// SIMATIC S7-200 project (STEP 7-Micro/WIN), CPU 226 CN REL 02.01

SYMBOL_TABLE 用户定义1
系统年              VW1648
本班开始运行小时         VW1680
本班开始运行分钟         VW1684
本班开始运行秒          VW1688
本班运行日            VW3778
系统日              VW1652
系统秒              VW1664
EEPROM写入次数       VW3558
累计运行分钟           VW1624
EEPROM写入后对秒脉冲计   VW3368
累计运行小时           VW1620
EEPROM写入后计时      M30.1
EEPROM传送中        SM31.7
SA2              I0.0     // 联锁/单独(单独=0/联锁=1)
PH1              I0.1     // 第1段线体首光电开关
PH11             I0.2     // 第1段线体末光电开关
PH2              I0.3     // 第2段线体首光电开关
PH21             I0.4     // 第2段线体末光电开关
PH3              I0.5     // 第3段线体首光电开关
PH31             I0.6     // 第3段线体末光电开关
PH4              I0.7     // 第4段线体首光电开关
PH41             I1.0     // 第4段线体末光电开关
PH5              I1.1     // 第5段线体首光电开关
PH6              I1.2     // 第6段线体末光电开关
PH7              I1.3     // 第7段线体首光电开关
PH71             I1.4     // 第7段线体末光电开关
PH8              I1.5     // 第8段线体首光电开关
PH9              I1.6     // 第9段线体末光电开关
PH10             I1.7     // 第10段线体首光电开关
PH101            I2.0     // 第10段线体末光电开关
SF1_SF11         I2.1     // 第1段线体启动
SJ1_SJ11         I2.2     // 第1段线体停止
SF2_SF21         I2.3     // 第2段线体启动
SJ2_SJ21         I2.4     // 第2段线体停止
SF3_SF31         I2.5     // 第3段线体启动
SJ3_SJ31         I2.6     // 第3段线体停止
SF4_SF41         I2.7     // 第4段线体启动
SJ4_SJ41         I3.0     // 第4段线体停止
SF5              I3.1     // 第5段线体启动
SJ5              I3.2     // 第5段线体停止
SF6              I3.3     // 第6段线体启动
SJ6              I3.4     // 第6段线体停止
SF7_SF71         I3.5     // 第8段线体启动
SJ7_SJ71         I3.6     // 第7段线体停止
SF8              I3.7     // 第8段线体启动
SJ8              I4.0     // 第8段线体停止
SF9              I4.1     // 第9段线体启动
SJ9              I4.2     // 第9段线体停止
SF10_SF101       I4.3     // 第10段线体启动
SJ10_SJ101       I4.4     // 第10段线体停止
SF110            I4.5     // 线体联锁启动
SS110            I4.6     // 线体联锁停止
SJ110            I4.7     // 全部停止
联锁运行             M0.0
联锁启动信号           M0.1
联锁停止信号           M0.2
电机全部停止           M0.3
PH11上升沿          M1.0
第一段线体就地启动        M1.1
PH21上升沿          M2.0
第二段线体就地启动        M2.1
PH31上升沿          M3.0
第三段线体就地启动        M3.1
PH41上升沿          M4.0
第四段线体就地启动        M4.1
PH5上升沿           M5.0
PH5动作保持          M5.1
PH6上升沿           M6.0
第5_6段线体就地启动      M6.1
PH71上升沿          M7.0
第七段线体就地启动        M7.1
PH8上升沿           M8.0
PH8动作保持          M8.1
PH9上升沿           M9.0
第8_9段线体就地启动      M9.1
PH101上升沿         M10.0
第十段线体就地启动        M10.1
上班时间             M31.4
HA1              Q0.0     // 启动告警
KA1              Q0.1     // 第1段线体电机M1
KA2              Q0.2     // 第2段线体电机M2
KA3              Q0.3     // 第3段线体电机M3
KA4              Q0.4     // 第4段线体电机M4
KA5              Q0.5     // 第5段线体电机M5
KA6              Q0.6     // 第6段线体电机M6
KA7              Q0.7     // 第7段线体电机M7
KA8              Q1.0     // 第8段线体电机M8
KA9              Q1.1     // 第9段线体电机M9
KA10             Q1.2     // 第10段线体电机M10
KA11             Q1.3     // 设备运行信号
HB1              Q1.4     // 单独/联锁指示(单独=0/联锁=1)
常ON标志位           SM0.0
秒时钟              SM0.5    // 0.5秒为1，0.5秒为0
启动告警时间           T37
第一段线体持续运行时间      T38
第二段线体持续运行时间      T39
第四段线体持续运行时间      T41
PH5动作后计时         T42
第5_6段线体持续运行时间    T43
第七段线体持续运行时间      T44
PH8动作后计时         T45
第8_9段线体持续运行时间    T46
第十段线体持续运行时间      T47
系统小时             VW1656
系统分钟             VW1660
上班小时             VW1720
上班分钟             VW1724
下班小时             VW1740
下班分钟             VW1744
END_SYMBOL_TABLE

ORGANIZATION_BLOCK 程序块:OB1
TITLE=华为技术有限公司天线装配线PLC程序
BEGIN
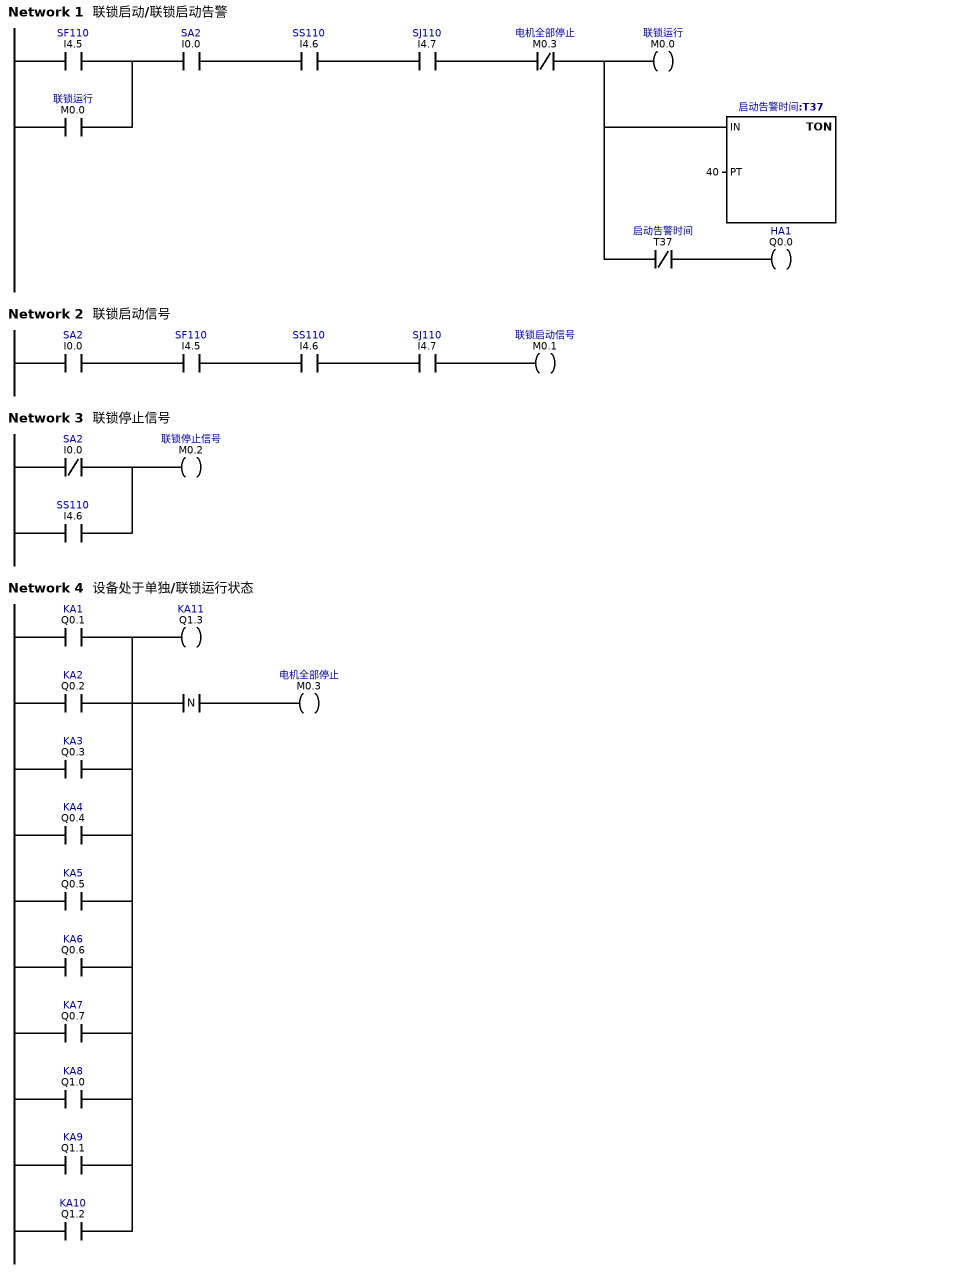
Network 1 // 联锁启动/联锁启动告警
LD     SF110:I4.5
O      联锁运行:M0.0
A      SA2:I0.0
A      SS110:I4.6
A      SJ110:I4.7
AN     电机全部停止:M0.3
=      联锁运行:M0.0
TON    启动告警时间:T37, 40
AN     启动告警时间:T37
=      HA1:Q0.0
Network 2 // 联锁启动信号
LD     SA2:I0.0
A      SF110:I4.5
A      SS110:I4.6
A      SJ110:I4.7
=      联锁启动信号:M0.1
Network 3 // 联锁停止信号
LDN    SA2:I0.0
O      SS110:I4.6
=      联锁停止信号:M0.2
Network 4 // 设备处于单独/联锁运行状态
LD     KA1:Q0.1
O      KA2:Q0.2
O      KA3:Q0.3
O      KA4:Q0.4
O      KA5:Q0.5
O      KA6:Q0.6
O      KA7:Q0.7
O      KA8:Q1.0
O      KA9:Q1.1
O      KA10:Q1.2
=      KA11:Q1.3
ED
=      电机全部停止:M0.3
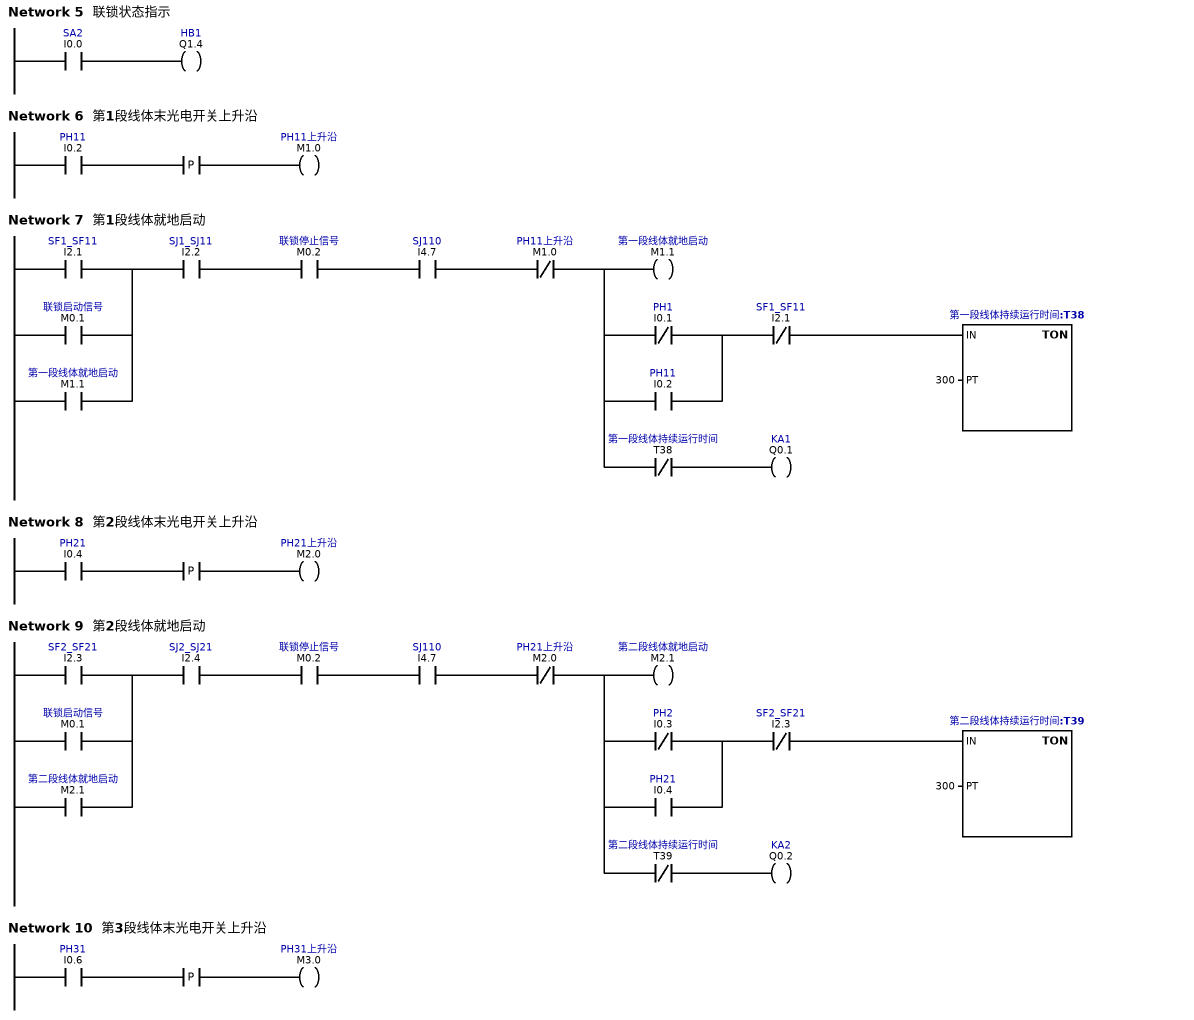
Network 5 // 联锁状态指示
LD     SA2:I0.0
=      HB1:Q1.4
Network 6 // 第1段线体末光电开关上升沿
LD     PH11:I0.2
EU
=      PH11上升沿:M1.0
Network 7 // 第1段线体就地启动
LD     SF1_SF11:I2.1
O      联锁启动信号:M0.1
O      第一段线体就地启动:M1.1
A      SJ1_SJ11:I2.2
A      联锁停止信号:M0.2
A      SJ110:I4.7
AN     PH11上升沿:M1.0
LPS
=      第一段线体就地启动:M1.1
LDN    PH1:I0.1
O      PH11:I0.2
ALD
AN     SF1_SF11:I2.1
TON    第一段线体持续运行时间:T38, 300
LPP
AN     第一段线体持续运行时间:T38
=      KA1:Q0.1
Network 8 // 第2段线体末光电开关上升沿
LD     PH21:I0.4
EU
=      PH21上升沿:M2.0
Network 9 // 第2段线体就地启动
LD     SF2_SF21:I2.3
O      联锁启动信号:M0.1
O      第二段线体就地启动:M2.1
A      SJ2_SJ21:I2.4
A      联锁停止信号:M0.2
A      SJ110:I4.7
AN     PH21上升沿:M2.0
LPS
=      第二段线体就地启动:M2.1
LDN    PH2:I0.3
O      PH21:I0.4
ALD
AN     SF2_SF21:I2.3
TON    第二段线体持续运行时间:T39, 300
LPP
AN     第二段线体持续运行时间:T39
=      KA2:Q0.2
Network 10 // 第3段线体末光电开关上升沿
LD     PH31:I0.6
EU
=      PH31上升沿:M3.0
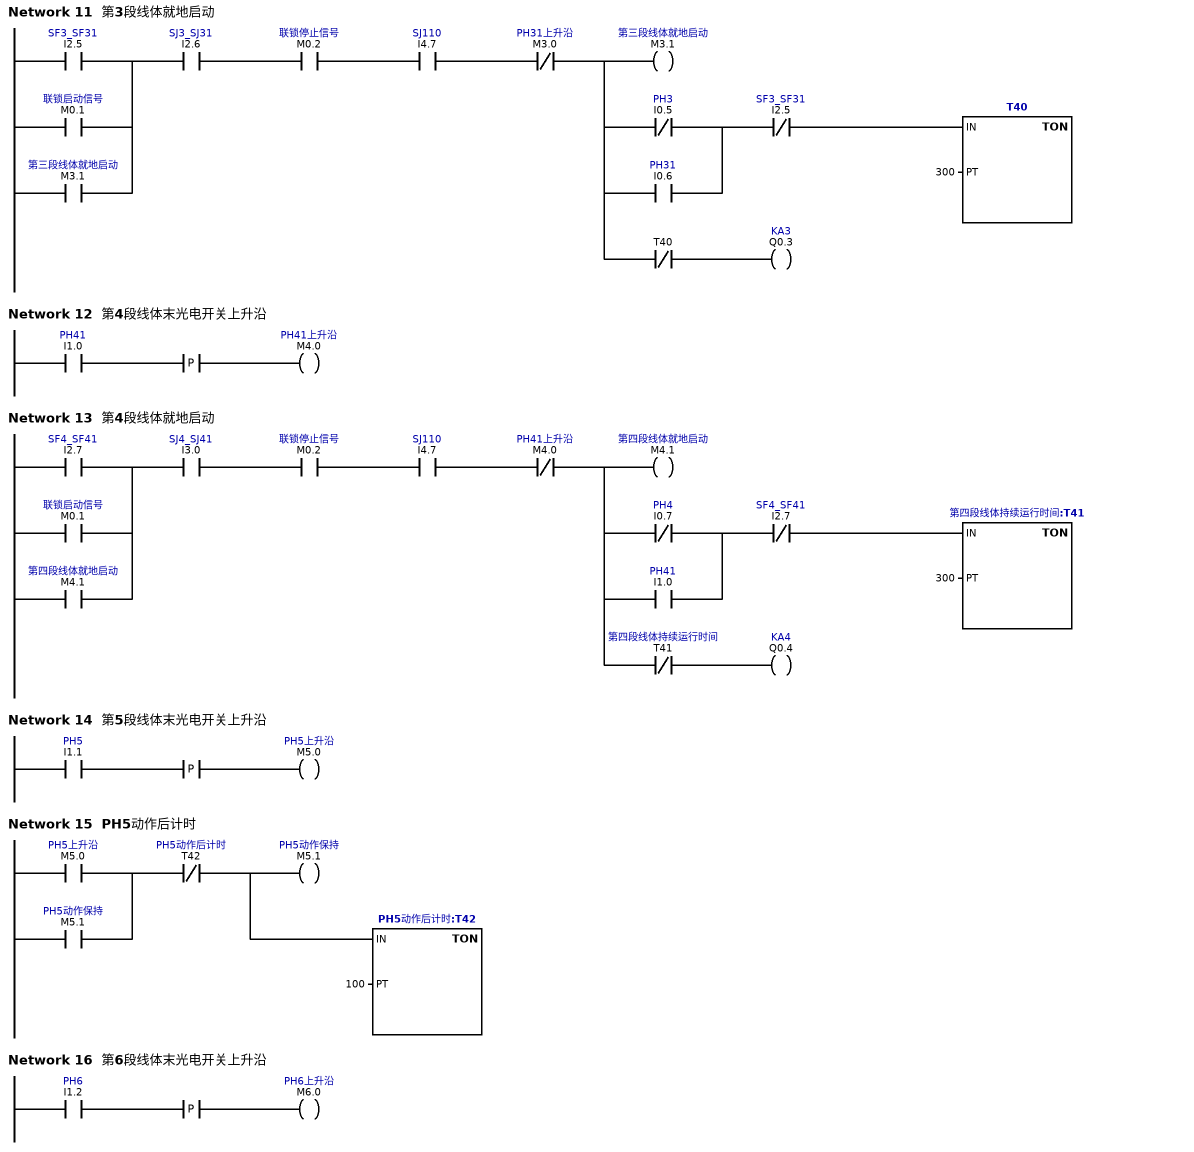
Network 11 // 第3段线体就地启动
LD     SF3_SF31:I2.5
O      联锁启动信号:M0.1
O      第三段线体就地启动:M3.1
A      SJ3_SJ31:I2.6
A      联锁停止信号:M0.2
A      SJ110:I4.7
AN     PH31上升沿:M3.0
LPS
=      第三段线体就地启动:M3.1
LDN    PH3:I0.5
O      PH31:I0.6
ALD
AN     SF3_SF31:I2.5
TON    T40, 300
LPP
AN     T40
=      KA3:Q0.3
Network 12 // 第4段线体末光电开关上升沿
LD     PH41:I1.0
EU
=      PH41上升沿:M4.0
Network 13 // 第4段线体就地启动
LD     SF4_SF41:I2.7
O      联锁启动信号:M0.1
O      第四段线体就地启动:M4.1
A      SJ4_SJ41:I3.0
A      联锁停止信号:M0.2
A      SJ110:I4.7
AN     PH41上升沿:M4.0
LPS
=      第四段线体就地启动:M4.1
LDN    PH4:I0.7
O      PH41:I1.0
ALD
AN     SF4_SF41:I2.7
TON    第四段线体持续运行时间:T41, 300
LPP
AN     第四段线体持续运行时间:T41
=      KA4:Q0.4
Network 14 // 第5段线体末光电开关上升沿
LD     PH5:I1.1
EU
=      PH5上升沿:M5.0
Network 15 // PH5动作后计时
LD     PH5上升沿:M5.0
O      PH5动作保持:M5.1
AN     PH5动作后计时:T42
=      PH5动作保持:M5.1
TON    PH5动作后计时:T42, 100
Network 16 // 第6段线体末光电开关上升沿
LD     PH6:I1.2
EU
=      PH6上升沿:M6.0
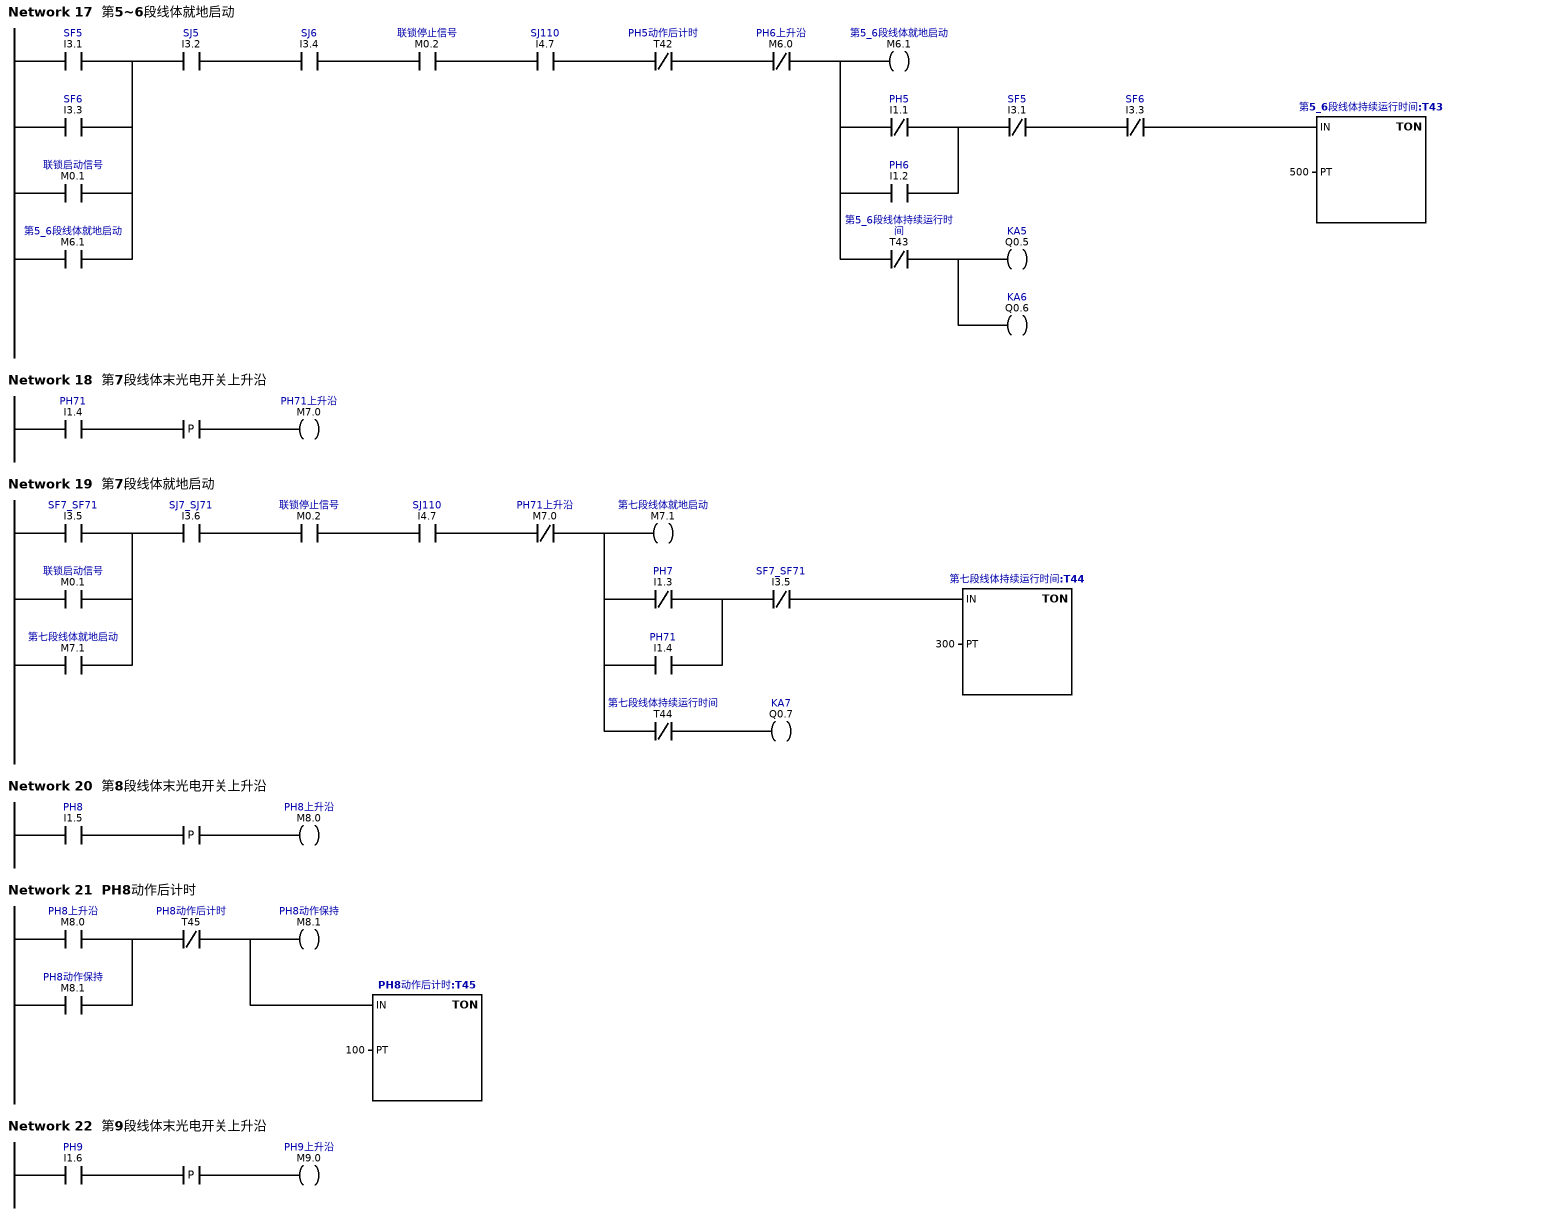
Network 17 // 第5~6段线体就地启动
LD     SF5:I3.1
O      SF6:I3.3
O      联锁启动信号:M0.1
O      第5_6段线体就地启动:M6.1
A      SJ5:I3.2
A      SJ6:I3.4
A      联锁停止信号:M0.2
A      SJ110:I4.7
AN     PH5动作后计时:T42
AN     PH6上升沿:M6.0
LPS
=      第5_6段线体就地启动:M6.1
LDN    PH5:I1.1
O      PH6:I1.2
ALD
AN     SF5:I3.1
AN     SF6:I3.3
TON    第5_6段线体持续运行时间:T43, 500
LPP
AN     第5_6段线体持续运行时间:T43
=      KA5:Q0.5
=      KA6:Q0.6
Network 18 // 第7段线体末光电开关上升沿
LD     PH71:I1.4
EU
=      PH71上升沿:M7.0
Network 19 // 第7段线体就地启动
LD     SF7_SF71:I3.5
O      联锁启动信号:M0.1
O      第七段线体就地启动:M7.1
A      SJ7_SJ71:I3.6
A      联锁停止信号:M0.2
A      SJ110:I4.7
AN     PH71上升沿:M7.0
LPS
=      第七段线体就地启动:M7.1
LDN    PH7:I1.3
O      PH71:I1.4
ALD
AN     SF7_SF71:I3.5
TON    第七段线体持续运行时间:T44, 300
LPP
AN     第七段线体持续运行时间:T44
=      KA7:Q0.7
Network 20 // 第8段线体末光电开关上升沿
LD     PH8:I1.5
EU
=      PH8上升沿:M8.0
Network 21 // PH8动作后计时
LD     PH8上升沿:M8.0
O      PH8动作保持:M8.1
AN     PH8动作后计时:T45
=      PH8动作保持:M8.1
TON    PH8动作后计时:T45, 100
Network 22 // 第9段线体末光电开关上升沿
LD     PH9:I1.6
EU
=      PH9上升沿:M9.0
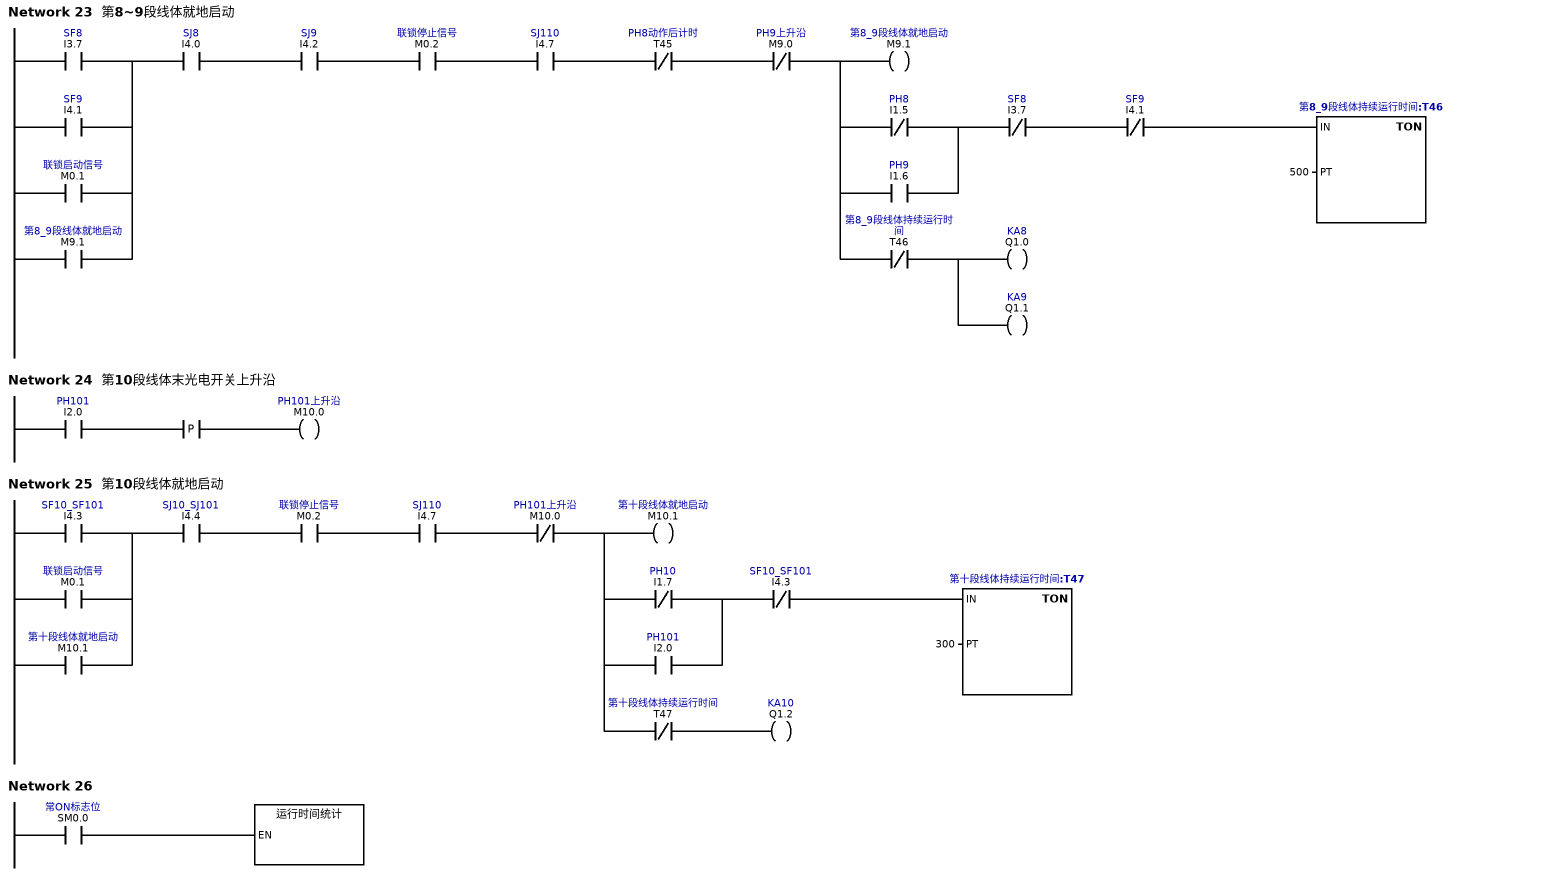
Network 23 // 第8~9段线体就地启动
LD     SF8:I3.7
O      SF9:I4.1
O      联锁启动信号:M0.1
O      第8_9段线体就地启动:M9.1
A      SJ8:I4.0
A      SJ9:I4.2
A      联锁停止信号:M0.2
A      SJ110:I4.7
AN     PH8动作后计时:T45
AN     PH9上升沿:M9.0
LPS
=      第8_9段线体就地启动:M9.1
LDN    PH8:I1.5
O      PH9:I1.6
ALD
AN     SF8:I3.7
AN     SF9:I4.1
TON    第8_9段线体持续运行时间:T46, 500
LPP
AN     第8_9段线体持续运行时间:T46
=      KA8:Q1.0
=      KA9:Q1.1
Network 24 // 第10段线体末光电开关上升沿
LD     PH101:I2.0
EU
=      PH101上升沿:M10.0
Network 25 // 第10段线体就地启动
LD     SF10_SF101:I4.3
O      联锁启动信号:M0.1
O      第十段线体就地启动:M10.1
A      SJ10_SJ101:I4.4
A      联锁停止信号:M0.2
A      SJ110:I4.7
AN     PH101上升沿:M10.0
LPS
=      第十段线体就地启动:M10.1
LDN    PH10:I1.7
O      PH101:I2.0
ALD
AN     SF10_SF101:I4.3
TON    第十段线体持续运行时间:T47, 300
LPP
AN     第十段线体持续运行时间:T47
=      KA10:Q1.2
Network 26
LD     常ON标志位:SM0.0
CALL   运行时间统计:SBR3
END_ORGANIZATION_BLOCK

// SBR1: protected block, not included

// SBR2: protected block, not included

SUBROUTINE_BLOCK 运行时间统计:SBR3
TITLE=运行时间统计程序
BEGIN
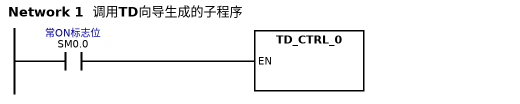
Network 1 // 调用TD向导生成的子程序
LD     常ON标志位:SM0.0
CALL   TD_CTRL_0:SBR1
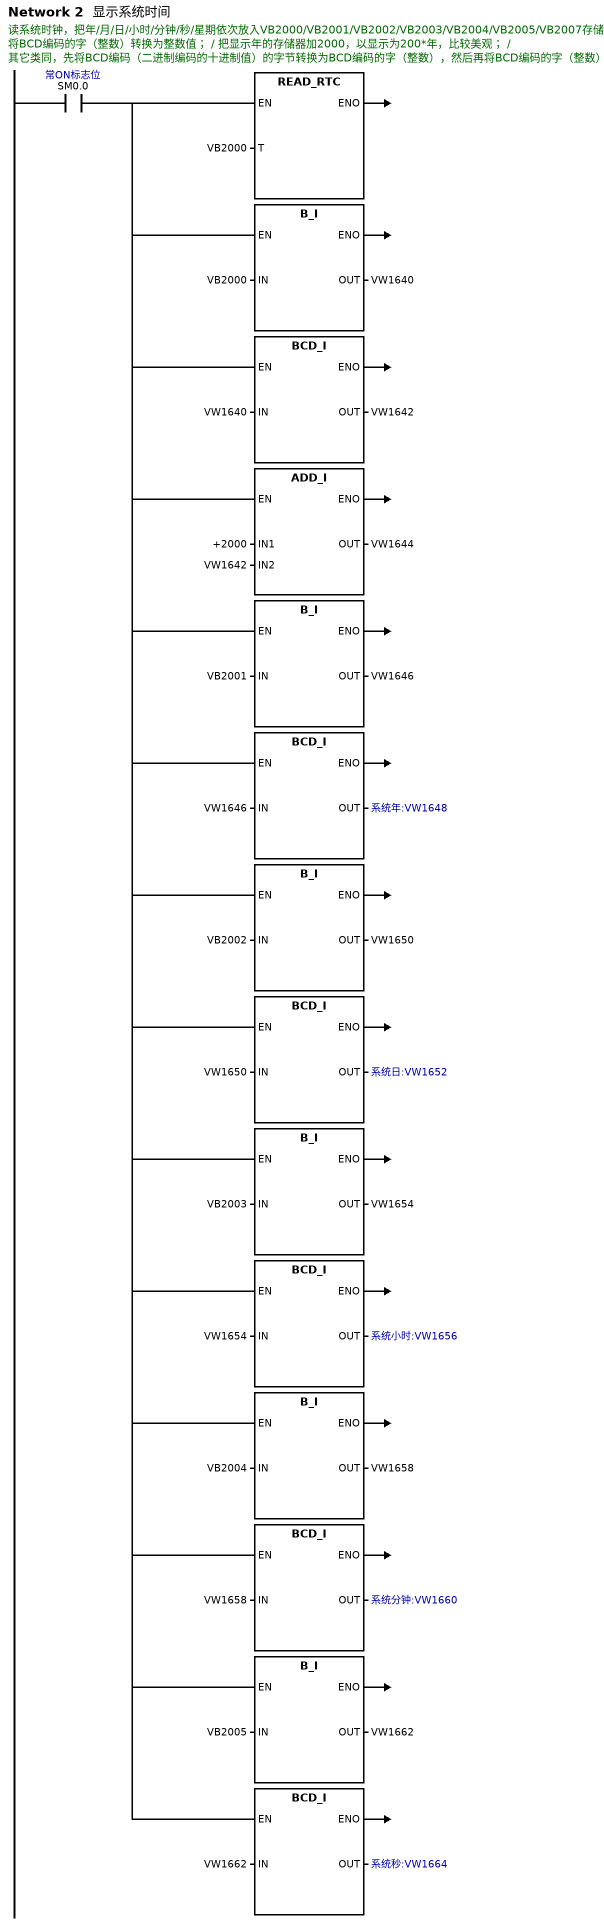
Network 2 // 显示系统时间
// 读系统时钟，把年/月/日/小时/分钟/秒/星期依次放入VB2000/VB2001/VB2002/VB2003/VB2004/VB2005/VB2007存储器中；
// 将BCD编码（二进制编码的十进制值）的字节转换为BCD编码的字（整数）；
// 将BCD编码的字（整数）转换为整数值；
// 把显示年的存储器加2000，以显示为200*年，比较美观；
// 其它类同，先将BCD编码（二进制编码的十进制值）的字节转换为BCD编码的字（整数），然后再将BCD编码的字（整数）转换为整数值；这样就得到了年/月/日/小时/分钟/秒的整数值（本程序没有处理星期，如果要处理，方法相同），以用于TD400C显示。
LD     常ON标志位:SM0.0
TODR   VB2000
BTI    VB2000, VW1640
MOVW   VW1640, VW1642
BCDI   VW1642
MOVW   +2000, VW1644
+I     VW1642, VW1644
BTI    VB2001, VW1646
MOVW   VW1646, 系统年:VW1648
BCDI   系统年:VW1648
BTI    VB2002, VW1650
MOVW   VW1650, 系统日:VW1652
BCDI   系统日:VW1652
BTI    VB2003, VW1654
MOVW   VW1654, 系统小时:VW1656
BCDI   系统小时:VW1656
BTI    VB2004, VW1658
MOVW   VW1658, 系统分钟:VW1660
BCDI   系统分钟:VW1660
BTI    VB2005, VW1662
MOVW   VW1662, 系统秒:VW1664
BCDI   系统秒:VW1664
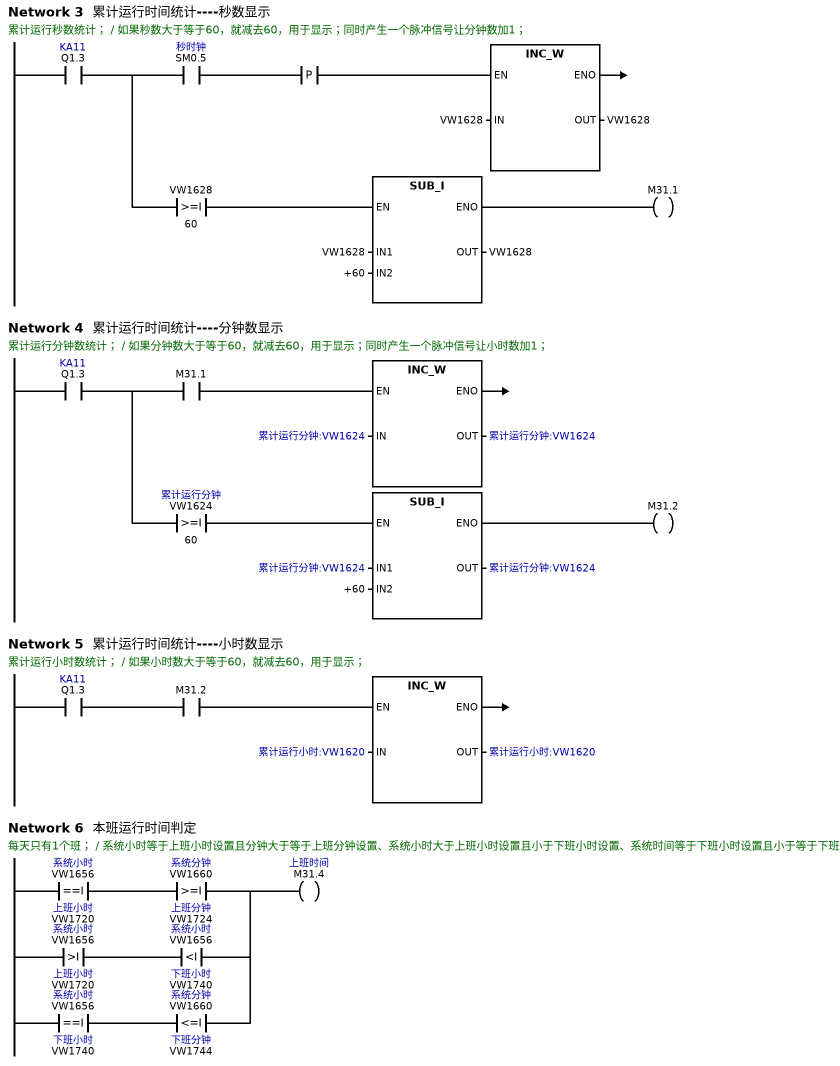
Network 3 // 累计运行时间统计----秒数显示
// 累计运行秒数统计；
// 如果秒数大于等于60，就减去60，用于显示；同时产生一个脉冲信号让分钟数加1；
LD     KA11:Q1.3
LPS
A      秒时钟:SM0.5
EU
INCW   VW1628
LPP
AW>=   VW1628, 60
-I     +60, VW1628
AENO
=      M31.1
Network 4 // 累计运行时间统计----分钟数显示
// 累计运行分钟数统计；
// 如果分钟数大于等于60，就减去60，用于显示；同时产生一个脉冲信号让小时数加1；
LD     KA11:Q1.3
LPS
A      M31.1
INCW   累计运行分钟:VW1624
LPP
AW>=   累计运行分钟:VW1624, 60
-I     +60, 累计运行分钟:VW1624
AENO
=      M31.2
Network 5 // 累计运行时间统计----小时数显示
// 累计运行小时数统计；
// 如果小时数大于等于60，就减去60，用于显示；
LD     KA11:Q1.3
A      M31.2
INCW   累计运行小时:VW1620
Network 6 // 本班运行时间判定
// 每天只有1个班；
// 系统小时等于上班小时设置且分钟大于等于上班分钟设置、系统小时大于上班小时设置且小于下班小时设置、系统时间等于下班小时设置且小于等于下班分钟设置，则认为是上班时间。
LDW=   系统小时:VW1656, 上班小时:VW1720
AW>=   系统分钟:VW1660, 上班分钟:VW1724
LDW>   系统小时:VW1656, 上班小时:VW1720
AW<    系统小时:VW1656, 下班小时:VW1740
OLD
LDW=   系统小时:VW1656, 下班小时:VW1740
AW<=   系统分钟:VW1660, 下班分钟:VW1744
OLD
=      上班时间:M31.4
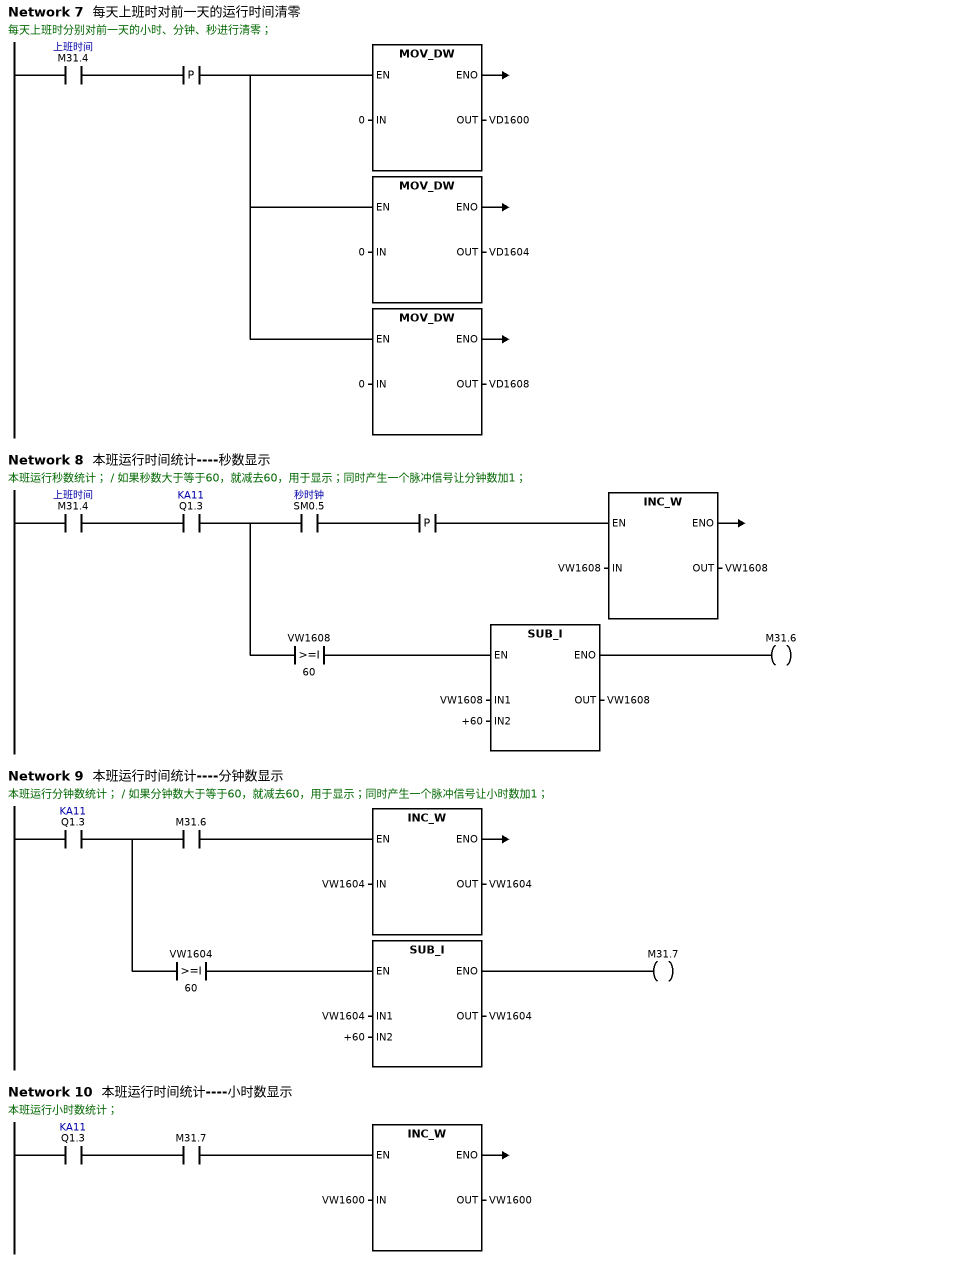
Network 7 // 每天上班时对前一天的运行时间清零
// 每天上班时分别对前一天的小时、分钟、秒进行清零；
LD     上班时间:M31.4
EU
MOVD   0, VD1600
MOVD   0, VD1604
MOVD   0, VD1608
Network 8 // 本班运行时间统计----秒数显示
// 本班运行秒数统计；
// 如果秒数大于等于60，就减去60，用于显示；同时产生一个脉冲信号让分钟数加1；
LD     上班时间:M31.4
A      KA11:Q1.3
LPS
A      秒时钟:SM0.5
EU
INCW   VW1608
LPP
AW>=   VW1608, 60
-I     +60, VW1608
AENO
=      M31.6
Network 9 // 本班运行时间统计----分钟数显示
// 本班运行分钟数统计；
// 如果分钟数大于等于60，就减去60，用于显示；同时产生一个脉冲信号让小时数加1；
LD     KA11:Q1.3
LPS
A      M31.6
INCW   VW1604
LPP
AW>=   VW1604, 60
-I     +60, VW1604
AENO
=      M31.7
Network 10 // 本班运行时间统计----小时数显示
// 本班运行小时数统计；
LD     KA11:Q1.3
A      M31.7
INCW   VW1600
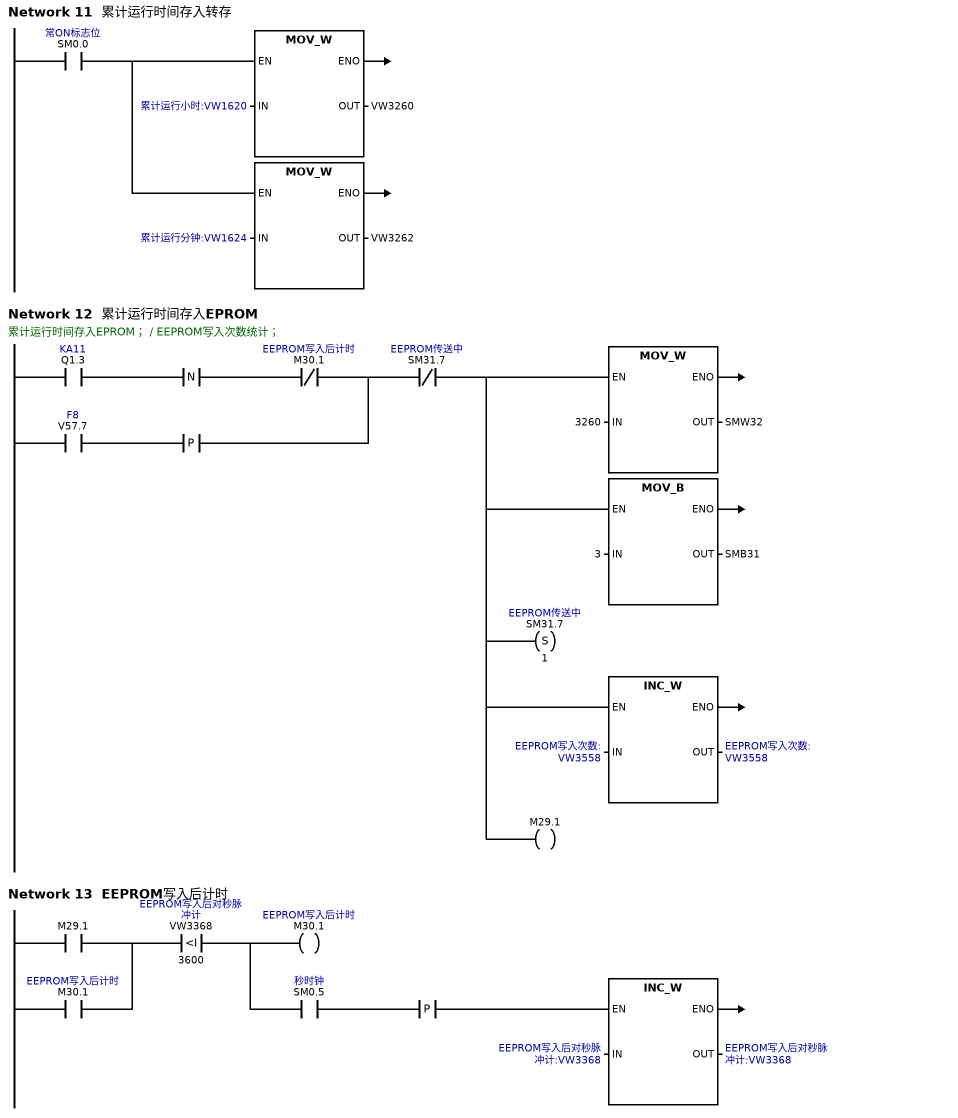
Network 11 // 累计运行时间存入转存
LD     常ON标志位:SM0.0
MOVW   累计运行小时:VW1620, VW3260
MOVW   累计运行分钟:VW1624, VW3262
Network 12 // 累计运行时间存入EPROM
// 累计运行时间存入EPROM；
// EEPROM写入次数统计；
LD     KA11:Q1.3
ED
AN     EEPROM写入后计时:M30.1
LD     F8:V57.7
EU
OLD
AN     EEPROM传送中:SM31.7
MOVW   3260, SMW32
MOVB   3, SMB31
S      EEPROM传送中:SM31.7, 1
INCW   EEPROM写入次数:VW3558
=      M29.1
Network 13 // EEPROM写入后计时
LD     M29.1
O      EEPROM写入后计时:M30.1
AW<    EEPROM写入后对秒脉冲计:VW3368, 3600
=      EEPROM写入后计时:M30.1
A      秒时钟:SM0.5
EU
INCW   EEPROM写入后对秒脉冲计:VW3368
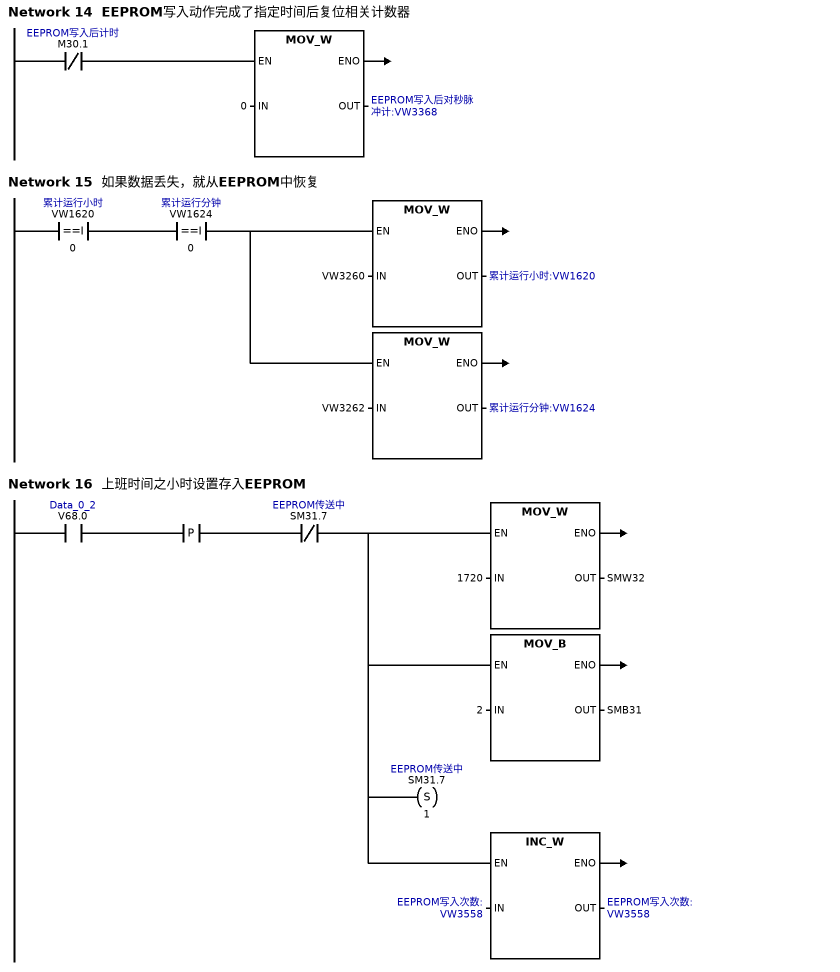
Network 14 // EEPROM写入动作完成了指定时间后复位相关计数器
LDN    EEPROM写入后计时:M30.1
MOVW   0, EEPROM写入后对秒脉冲计:VW3368
Network 15 // 如果数据丢失，就从EEPROM中恢复
LDW=   累计运行小时:VW1620, 0
AW=    累计运行分钟:VW1624, 0
MOVW   VW3260, 累计运行小时:VW1620
MOVW   VW3262, 累计运行分钟:VW1624
Network 16 // 上班时间之小时设置存入EEPROM
LD     Data_0_2:V68.0
EU
AN     EEPROM传送中:SM31.7
MOVW   1720, SMW32
MOVB   2, SMB31
S      EEPROM传送中:SM31.7, 1
INCW   EEPROM写入次数:VW3558
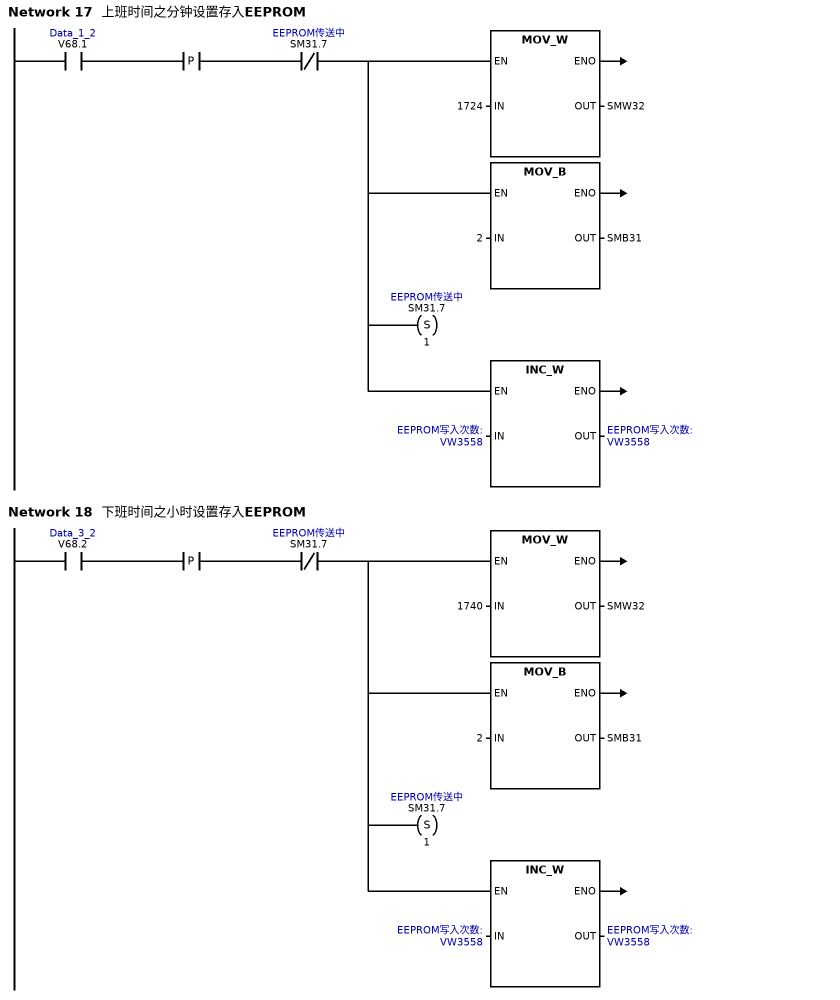
Network 17 // 上班时间之分钟设置存入EEPROM
LD     Data_1_2:V68.1
EU
AN     EEPROM传送中:SM31.7
MOVW   1724, SMW32
MOVB   2, SMB31
S      EEPROM传送中:SM31.7, 1
INCW   EEPROM写入次数:VW3558
Network 18 // 下班时间之小时设置存入EEPROM
LD     Data_3_2:V68.2
EU
AN     EEPROM传送中:SM31.7
MOVW   1740, SMW32
MOVB   2, SMB31
S      EEPROM传送中:SM31.7, 1
INCW   EEPROM写入次数:VW3558
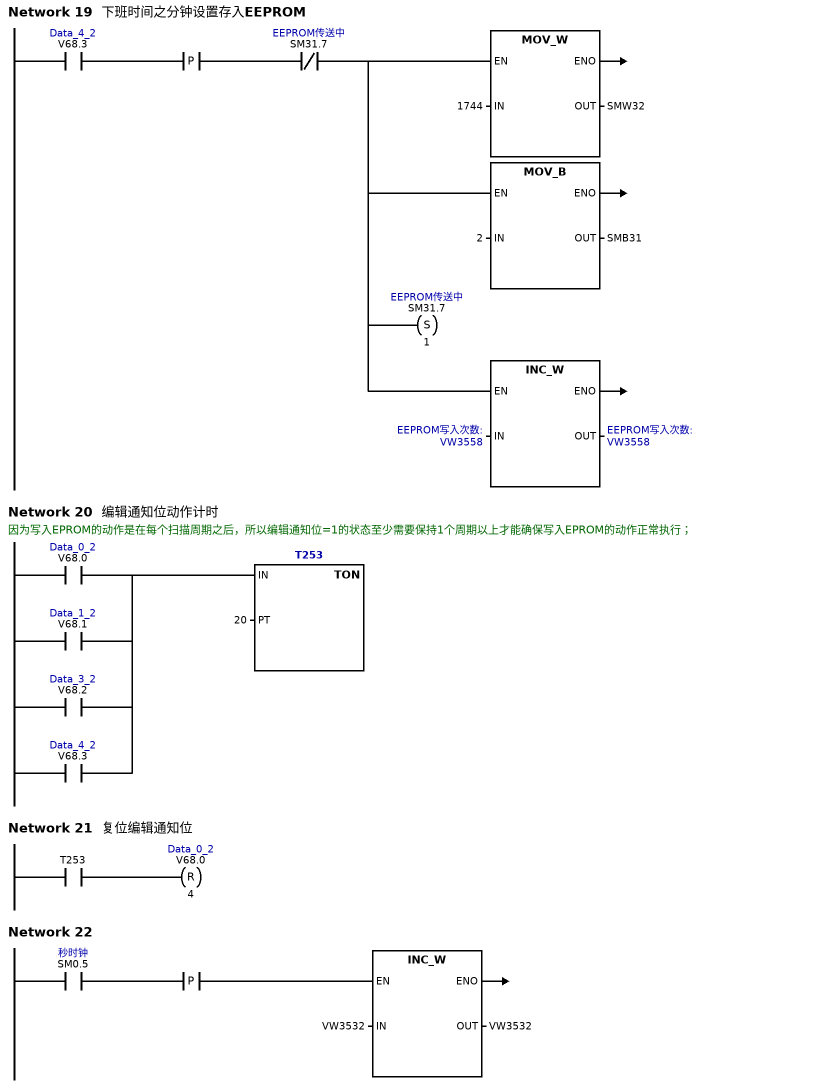
Network 19 // 下班时间之分钟设置存入EEPROM
LD     Data_4_2:V68.3
EU
AN     EEPROM传送中:SM31.7
MOVW   1744, SMW32
MOVB   2, SMB31
S      EEPROM传送中:SM31.7, 1
INCW   EEPROM写入次数:VW3558
Network 20 // 编辑通知位动作计时
// 因为写入EPROM的动作是在每个扫描周期之后，所以编辑通知位=1的状态至少需要保持1个周期以上才能确保写入EPROM的动作正常执行；
LD     Data_0_2:V68.0
O      Data_1_2:V68.1
O      Data_3_2:V68.2
O      Data_4_2:V68.3
TON    T253, 20
Network 21 // 复位编辑通知位
LD     T253
R      Data_0_2:V68.0, 4
Network 22
LD     秒时钟:SM0.5
EU
INCW   VW3532
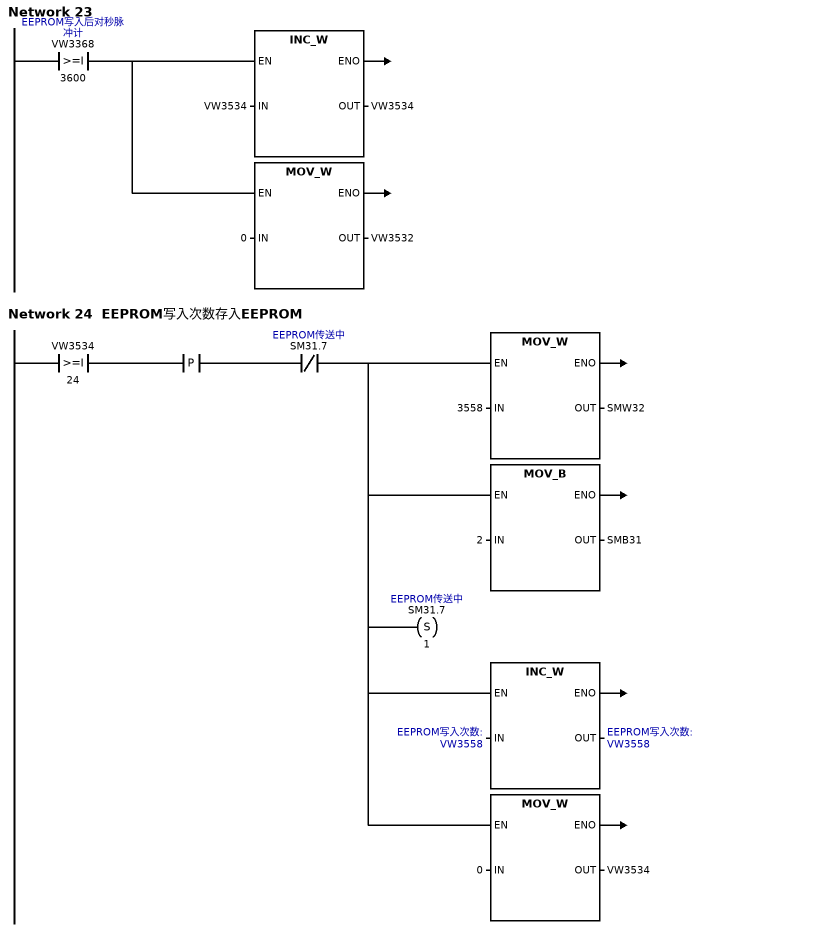
Network 23
LDW>=  EEPROM写入后对秒脉冲计:VW3368, 3600
INCW   VW3534
MOVW   0, VW3532
Network 24 // EEPROM写入次数存入EEPROM
LDW>=  VW3534, 24
EU
AN     EEPROM传送中:SM31.7
MOVW   3558, SMW32
MOVB   2, SMB31
S      EEPROM传送中:SM31.7, 1
INCW   EEPROM写入次数:VW3558
MOVW   0, VW3534
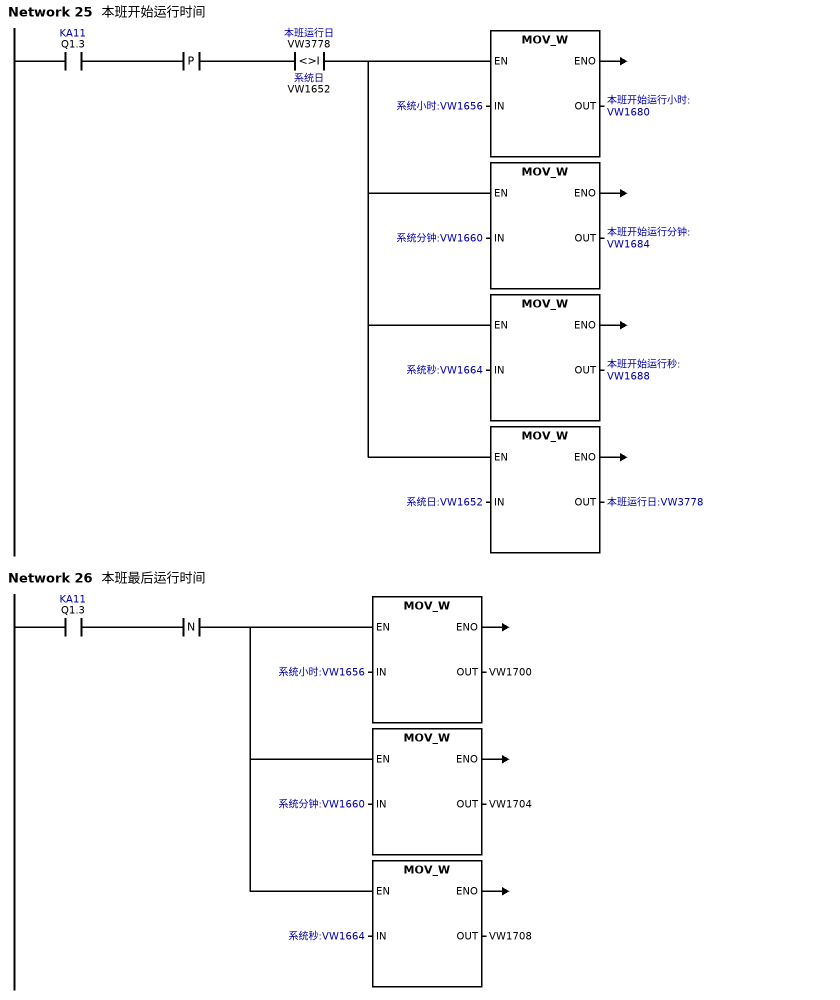
Network 25 // 本班开始运行时间
LD     KA11:Q1.3
EU
AW<>   本班运行日:VW3778, 系统日:VW1652
MOVW   系统小时:VW1656, 本班开始运行小时:VW1680
MOVW   系统分钟:VW1660, 本班开始运行分钟:VW1684
MOVW   系统秒:VW1664, 本班开始运行秒:VW1688
MOVW   系统日:VW1652, 本班运行日:VW3778
Network 26 // 本班最后运行时间
LD     KA11:Q1.3
ED
MOVW   系统小时:VW1656, VW1700
MOVW   系统分钟:VW1660, VW1704
MOVW   系统秒:VW1664, VW1708
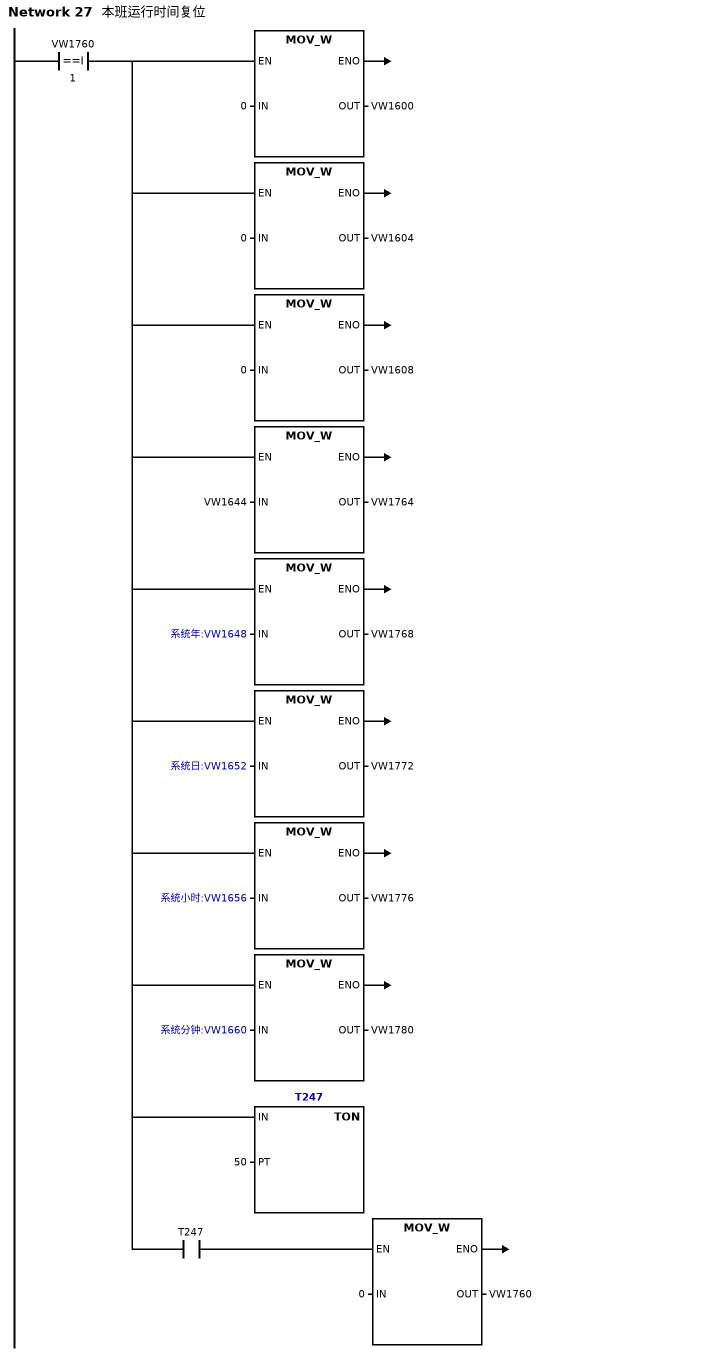
Network 27 // 本班运行时间复位
LDW=   VW1760, 1
MOVW   0, VW1600
MOVW   0, VW1604
MOVW   0, VW1608
MOVW   VW1644, VW1764
MOVW   系统年:VW1648, VW1768
MOVW   系统日:VW1652, VW1772
MOVW   系统小时:VW1656, VW1776
MOVW   系统分钟:VW1660, VW1780
TON    T247, 50
A      T247
MOVW   0, VW1760
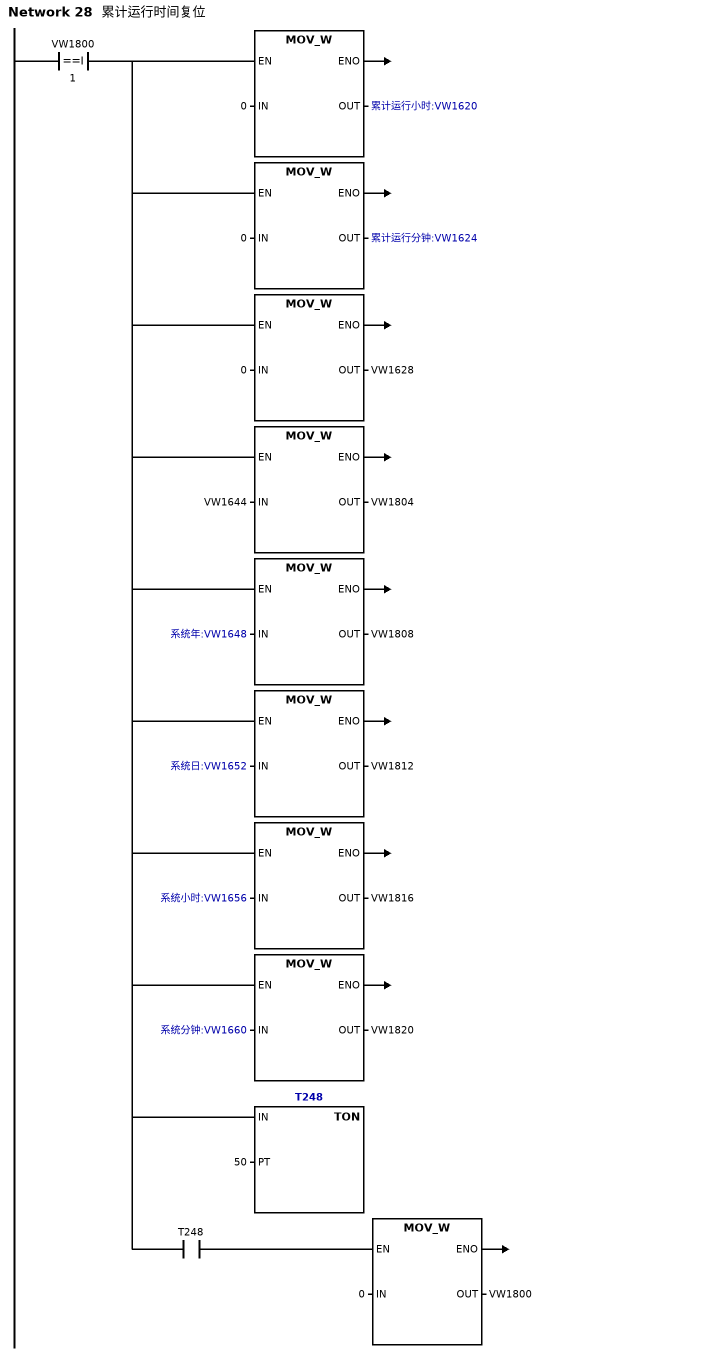
Network 28 // 累计运行时间复位
LDW=   VW1800, 1
MOVW   0, 累计运行小时:VW1620
MOVW   0, 累计运行分钟:VW1624
MOVW   0, VW1628
MOVW   VW1644, VW1804
MOVW   系统年:VW1648, VW1808
MOVW   系统日:VW1652, VW1812
MOVW   系统小时:VW1656, VW1816
MOVW   系统分钟:VW1660, VW1820
TON    T248, 50
A      T248
MOVW   0, VW1800
END_SUBROUTINE_BLOCK

// (further data pages could not be read)
